(* PLC project TEST.project, CODESYS CODESYS V3.5 SP3 Patch 7 *)
(* stored: creationDateTime 2013-12-18T19:09:11.7818395, modificationDateTime 2013-12-18T18:56:49.0513577 *)

FUNCTION_BLOCK Band
  VAR
    Motor : INT;
    links : INT;
    rechts : INT;
    Signal : INT;
    Ende : INT;
  END_VAR

INITIAL_STEP Band steht:
END_STEP
TRANSITION FROM Band steht TO Band vorwärts
  := Motor links;
END_TRANSITION
TRANSITION FROM Band steht TO Band rückwärts
  := Motor rechts;
END_TRANSITION
STEP Band vorwärts:
END_STEP
TRANSITION FROM Band vorwärts TO Init
  := Signal Ende;
END_TRANSITION
STEP Band rückwärts:
END_STEP
TRANSITION FROM Band rückwärts TO Init
  := Trans1;
END_TRANSITION
END_FUNCTION_BLOCK
